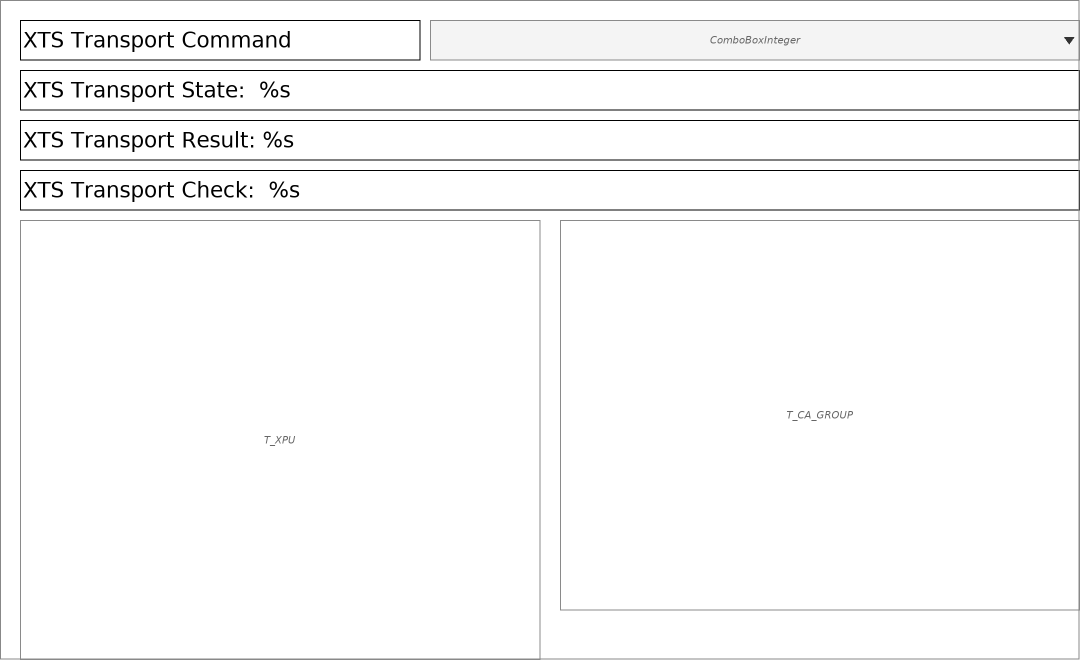
VISUALIZATION XTS_TRANSPORT_1  // 1080x660
    Rectangle (20,20 400x40), "XTS Transport Command"
    ComboBoxInteger (430,20 650x40), variable: GVL_XTS.XtsTransportCtrl.Cmd, text list: 'TL_E_CTRL_TRANSPORT'
    Rectangle (20,70 1060x40), "XTS Transport State: %s", text variable: MAIN_XTS.sTransportState
    Rectangle (20,120 1060x40), "XTS Transport Result: %s", text variable: MAIN_XTS.sTransportResult
    Rectangle (20,170 1060x40), "XTS Transport Check: %s", text variable: MAIN_XTS.sTransportCheck
    Frame (20,220 520x440)
        shows T_XPU(stXpuState := GVL_XTS.XtsTransportState.XpuState, stXpuInfo := GVL_XTS.XtsTransportState.XpuInfo, stXpuStrings := MAIN_XTS.stXpuStrings)
    Frame (560,220 520x390)
        shows T_CA_GROUP(stGroupInfo := GVL_XTS.XtsTransportState.GroupInfo, sGroupState := MAIN_XTS.sCaGroupState)
END_VISUALIZATION

(* stored: Version 1.1.0.1, ProductVersion 3.1.4026.20
   Visu XTS_TRANSPORT_1: Id {a5a6c3b0-7aa2-4848-86db-444d1e85ff6d} *)
